PROGRAM Winder_data
VAR
	Power_lever_0: Power_lever;
	Clutch_0: Clutch;
	TP_0: TP;
	Brake_0: Brake;
	Standard_stuff_0:Standard_stuff;
	TP_1: TP;
	TP_2: TP;
END_VAR
VAR // added by the converter: edge detectors and wires of the graphical bodies
    _w1, _w2, _w3, _w4, _w5 : ANY;
END_VAR

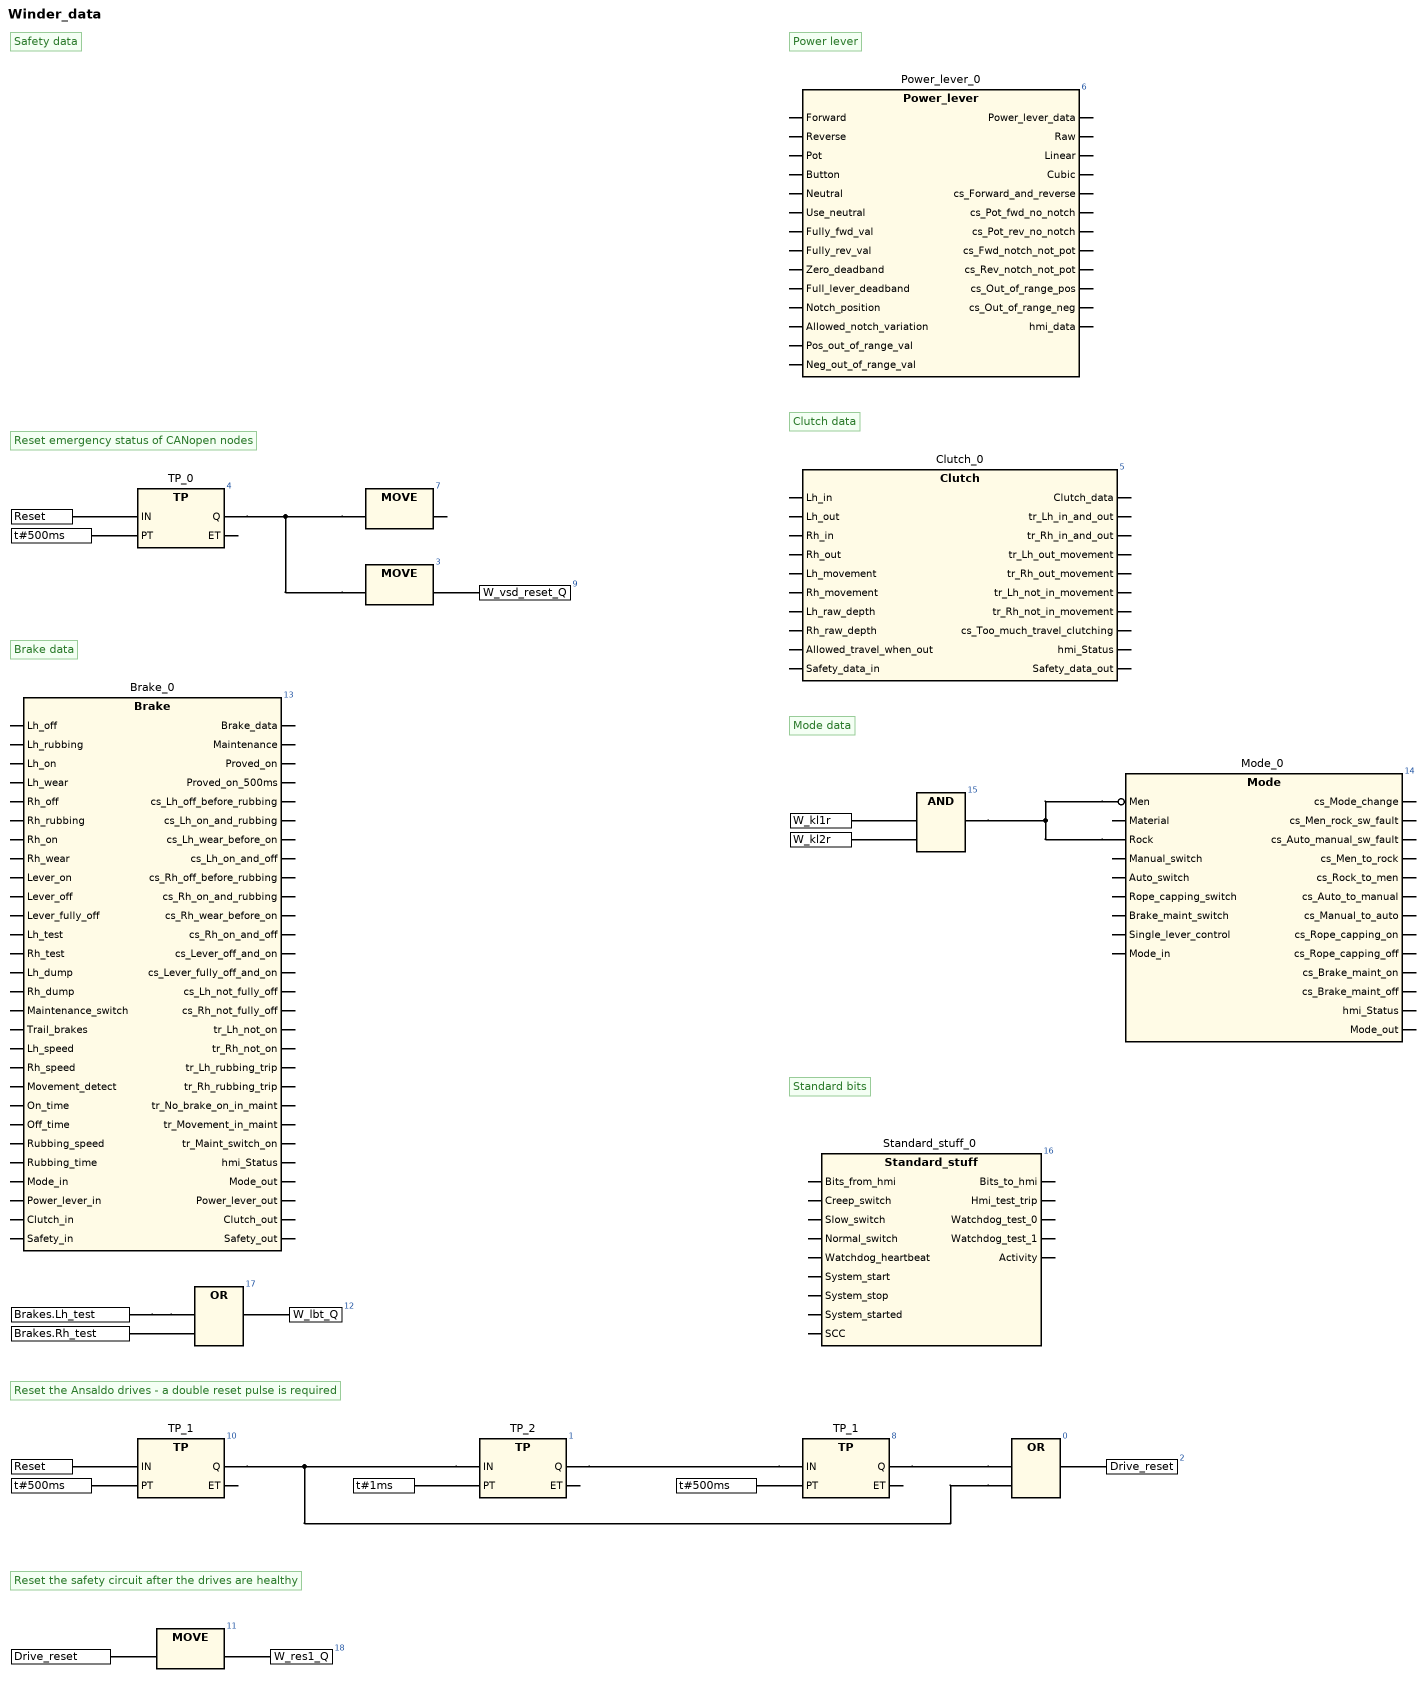
_w1 := TP_1.Q OR TP_1.Q;
TP_2(IN := TP_1.Q, PT := t#1ms); // TP
Drive_reset := _w1;
_w2 := TP_0.Q;
// Reset emergency status of CANopen nodes
TP_0(IN := Reset, PT := t#500ms); // TP
// Clutch data
Clutch_0(); // Clutch
// Safety data
// Power lever
Power_lever_0(); // Power_lever
(* TP_0.Q; result not used *)
TP_1(IN := TP_2.Q, PT := t#500ms); // TP
W_vsd_reset_Q := _w2;
// Reset the Ansaldo drives - a double reset pulse is required
TP_1(IN := Reset, PT := t#500ms); // TP
// Reset the safety circuit after the drives are healthy
_w3 := Drive_reset;
W_lbt_Q := _w4;
// Brake data
Brake_0(); // Brake
Mode_0(Men := NOT _w5, Rock := _w5); // Mode
// Mode data
_w5 := W_kl1r AND W_kl2r;
// Standard bits
Standard_stuff_0(); // Standard_stuff
_w4 := Brakes.Lh_test OR Brakes.Rh_test;
W_res1_Q := _w3;

METHOD Brake
VAR_INPUT
	Lh_off:BOOL;(*Left brake off signal - usually from left spring nest*)
	Lh_rubbing:BOOL; (*Left brake rubbing signal - usually from left spring nest*)
	Lh_on:BOOL; (*Left brake on signal - usually from left spring nest*)
	Lh_wear:BOOL; (*Left brake wear signal - usually from left spring nest*)
	Rh_off:BOOL; (*Right brake on signal - usually from right spring nest*)
	Rh_rubbing:BOOL; (*Right brake rubbing signal - usually from right spring nest*)
	Rh_on:BOOL; (*Right brake on signal - usually from right spring nest*)
	Rh_wear:BOOL; (*Right brake wear signal - usually from Right spring nest*)
	Lever_on:BOOL; (*Brake lever on limit switch*)
	Lever_off:BOOL; (*Brake lever off - normally from same limit switch as "Lever_on"*)
	Lever_fully_off:BOOL; (*Brake lever fully off limit switch. Necessary for automatic winders.*)
	Lh_test:BOOL; (*Left brake test switch - normally on driver's desk. Often the same switch as Lh_dump.*)
	Rh_test:BOOL; (*Right brake test switch - normally on driver's desk. Often the same switch as Rh_dump.*)
	Lh_dump:BOOL; (*Left brake dump switch - normally on driver's desk. Often the same switch as Lh_test.*)
	Rh_dump:BOOL; (*Right brake dump switch - normally on driver's desk. Often the same switch as Rh_test.*)
	Maintenance_switch:BOOL; (*Brake maintenance switch (can be on driver's desk or in control panels).*)
	Trail_brakes:BOOL; (*Trail brake control signal. Used to disable Lh_not_fully_off and Rh_not_fully_off trips.*)
	Lh_speed:INT; (*Left drum speed (normally in mm/s)*)
	Rh_speed:INT; (*Right drum speed (normally in mm/s)*)
	Movement_detect:BOOL; (*Drum movement detected (on either of the two drums in a double-drum winder)*)
	On_time:TIME; (*Maximum time allowed for brakes to apply.*)
	Off_time:TIME; (*Maximum time allowed for brakes to lift.*)
	Rubbing_speed:INT; (*Speed above which the brakes must be above the rubbing position*)
	Rubbing_time:TIME; (*Time before brake rubbing trips trigger *)
	Mode_in:dut_Mode;
	Power_lever_in:dut_Power_lever;
	Clutch_in:dut_Clutch;
	Safety_in:dut_Safety;
END_VAR
VAR_OUTPUT
	Brake_data:dut_Brake;
	Maintenance:BOOL; (*The winder is in brake maintenance mode*)
	Proved_on:BOOL; (*The brake lever (if in manual mode) and both brakes are on*)
	Proved_on_500ms:BOOL; (*The brakes have been proved on for 500ms*)
	cs_Lh_off_before_rubbing:BOOL; (*The Lh_off switch has closed but the Lh_rubbing switch has not yet closed*)
	cs_Lh_on_and_rubbing:BOOL; (*The Lh_on switch has closed but the Lh_rubbing switch is still closed*)
	cs_Lh_wear_before_on:BOOL; (*The Lh_on switch has closed but the Lh_rubbing switch is still closed*)
	cs_Lh_on_and_off:BOOL; (*The Lh_on and Lh_off switches are simultaneously closed*)
	cs_Rh_off_before_rubbing:BOOL; (*The Rh_off switch has closed but the Rh_rubbing switch has not yet closed*)
	cs_Rh_on_and_rubbing:BOOL; (*The Rh_on switch has closed but the Rh_rubbing switch is still closed*)
	cs_Rh_wear_before_on:BOOL; (*The Rh_on switch has closed but the Rh_rubbing switch is still closed*)
	cs_Rh_on_and_off:BOOL; (*The Rh_on and Rh_off switches are simultaneously closed*)
	cs_Lever_off_and_on:BOOL; (*The brake lever on and off switches are simultaneously closed*)
	cs_Lever_fully_off_and_on:BOOL; (*The brake lever on and fully off switches are simultaneously closed*)
	cs_Lh_not_fully_off:BOOL; (*The brake lever has been off for longer than the brake lift time but the Lh_off switch is not closed. Trail_brakes disables this fault.*)
	cs_Rh_not_fully_off:BOOL; (*The brake lever has been off for longer than the brake lift time but the Rh_off switch is not closed. Trail_brakes disables this fault.*)
	tr_Lh_not_on:BOOL; (*The brake lever has been on for longer than the brake application time but the Lh_on switch is not closed.*)
	tr_Rh_not_on:BOOL; (*The brake lever has been on for longer than the brake application time but the Rh_on switch is not closed.*)
	tr_Lh_rubbing_trip:BOOL; (*Lh_rubbing active above the rubbing trip speed*)
	tr_Rh_rubbing_trip:BOOL; (*Rh_rubbing active above the rubbing trip speed*)
	tr_No_brake_on_in_maint:BOOL; (*The power lever was moved from the neutral position in brake maintenance mode*)
	tr_Movement_in_maint:BOOL; (*Movement has been detected in brake maintenance mode*)
	tr_Maint_switch_on:BOOL; (*The brake maintenance switch is on but a brake is not dumped*)
	hmi_Status:ARRAY[1..2] OF WORD; (*Status bits for HMI*)
	Mode_out:dut_Mode;
	Power_lever_out:dut_Power_lever;
	Clutch_out:dut_Clutch;
	Safety_out:dut_Safety;
END_VAR
VAR
	TON_0: TON;
	Maintenance_req: BOOL;
	RS_0: RS;
	TON_1: TON;
	TON_2: TON;
	TON_3: TON;
	TON_4: TON;
	TON_5: TON;
	TON_6: TON;
	TON_7: TON;
	TON_8: TON;
	TON_9: TON;
	TON_10: TON;
	TON_11: TON;
	TON_12: TON;
	TON_13: TON;
	TON_14: TON;
	TON_15: TON;
	TON_16: TON;
	TON_17: TON;
END_VAR
VAR_INST // added by the converter: edge detectors and wires of the graphical bodies
    _w1, _w3, _w5, _w8, _w9, _w10, _w11, _w12, _w13, _w14, _w15, _w16, _w17, _w18, _w19, _w20, _w21, _w22, _w23, _w24, _w26, _w27, _w28 : BOOL;
    _w2, _w4, _w6, _w7, _w25 : ANY;
END_VAR
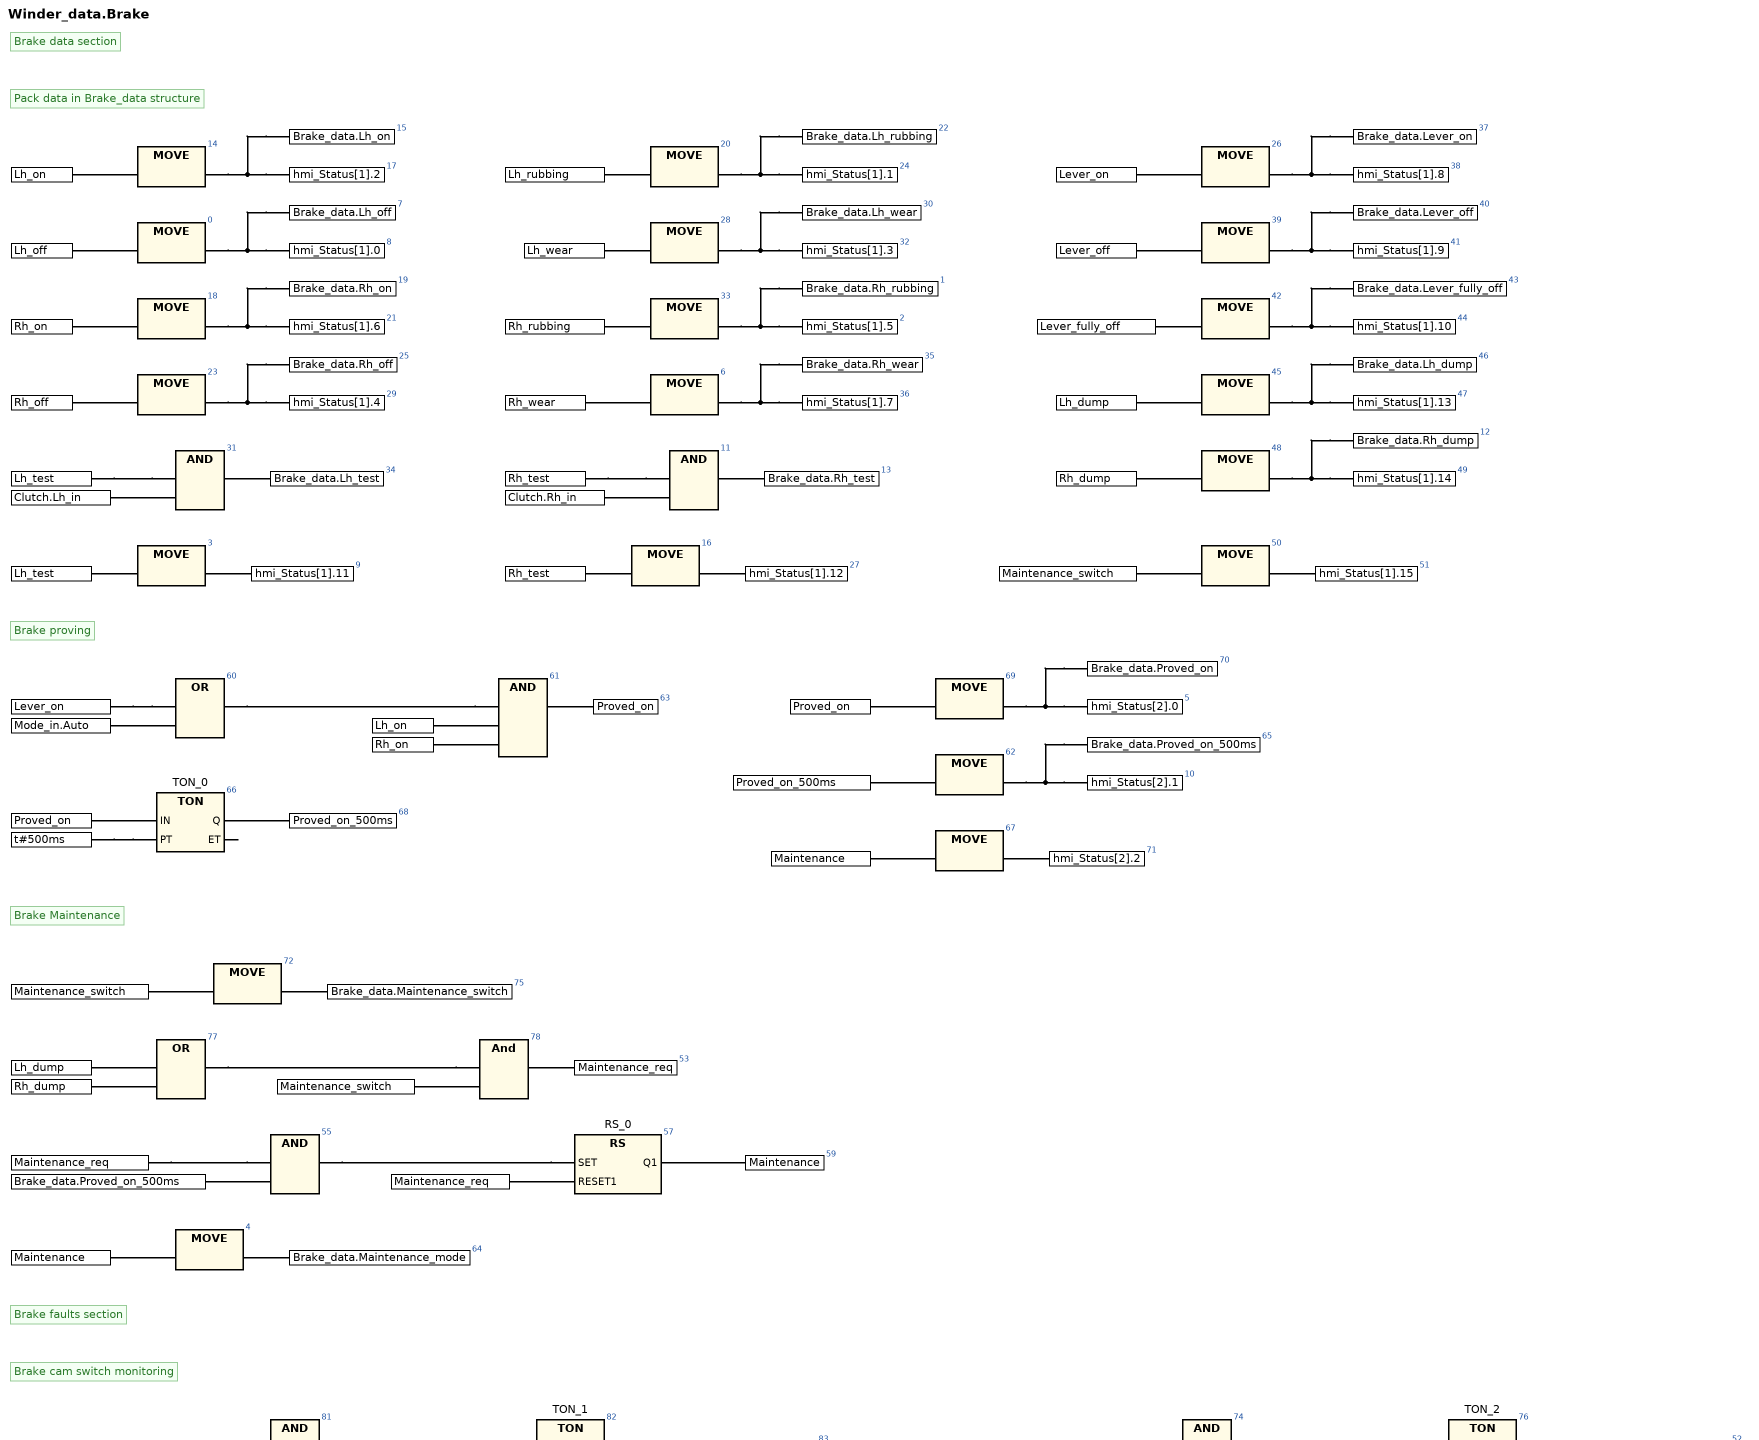
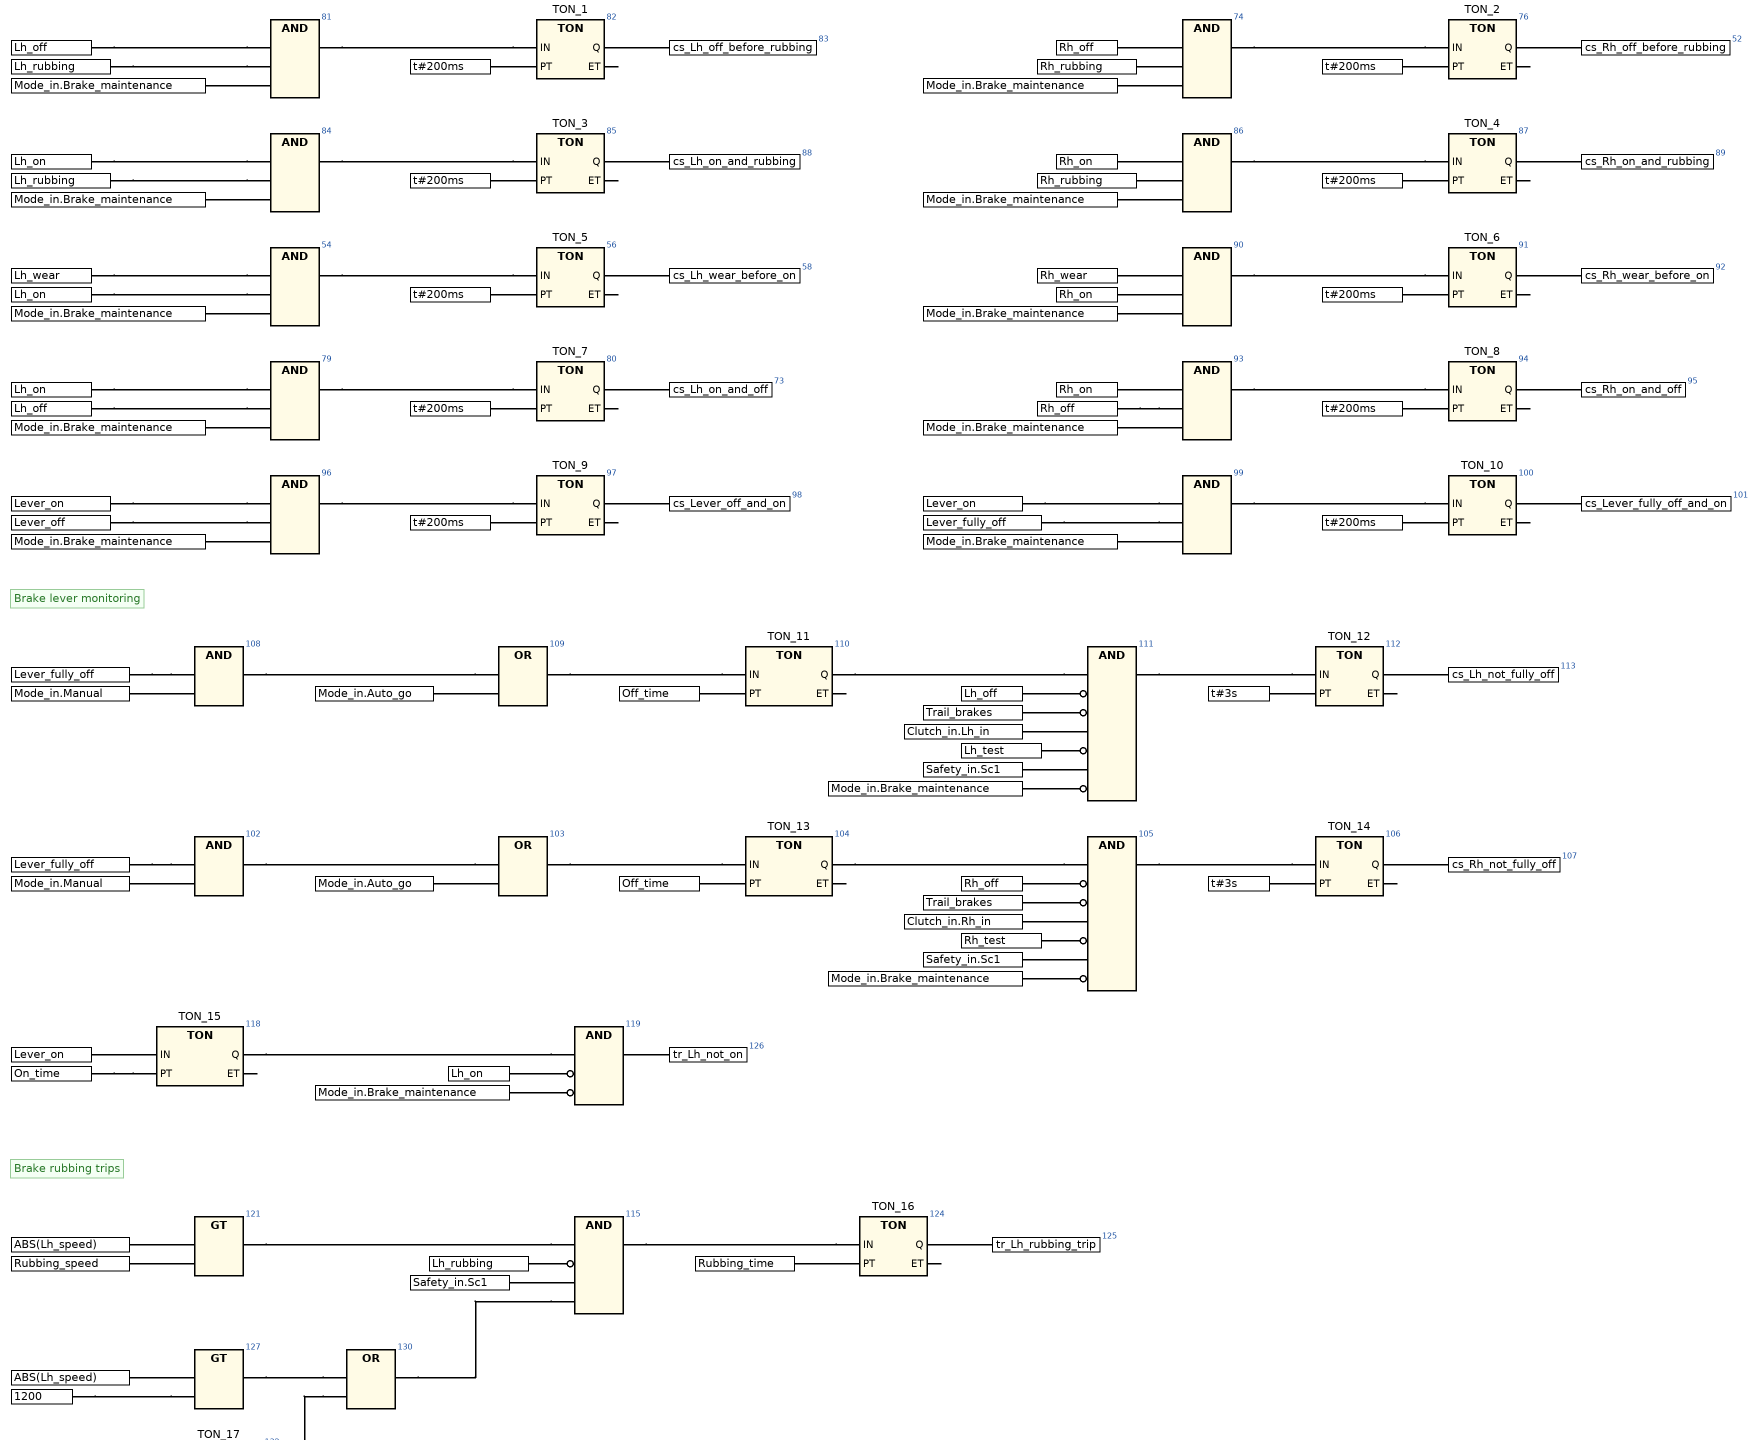
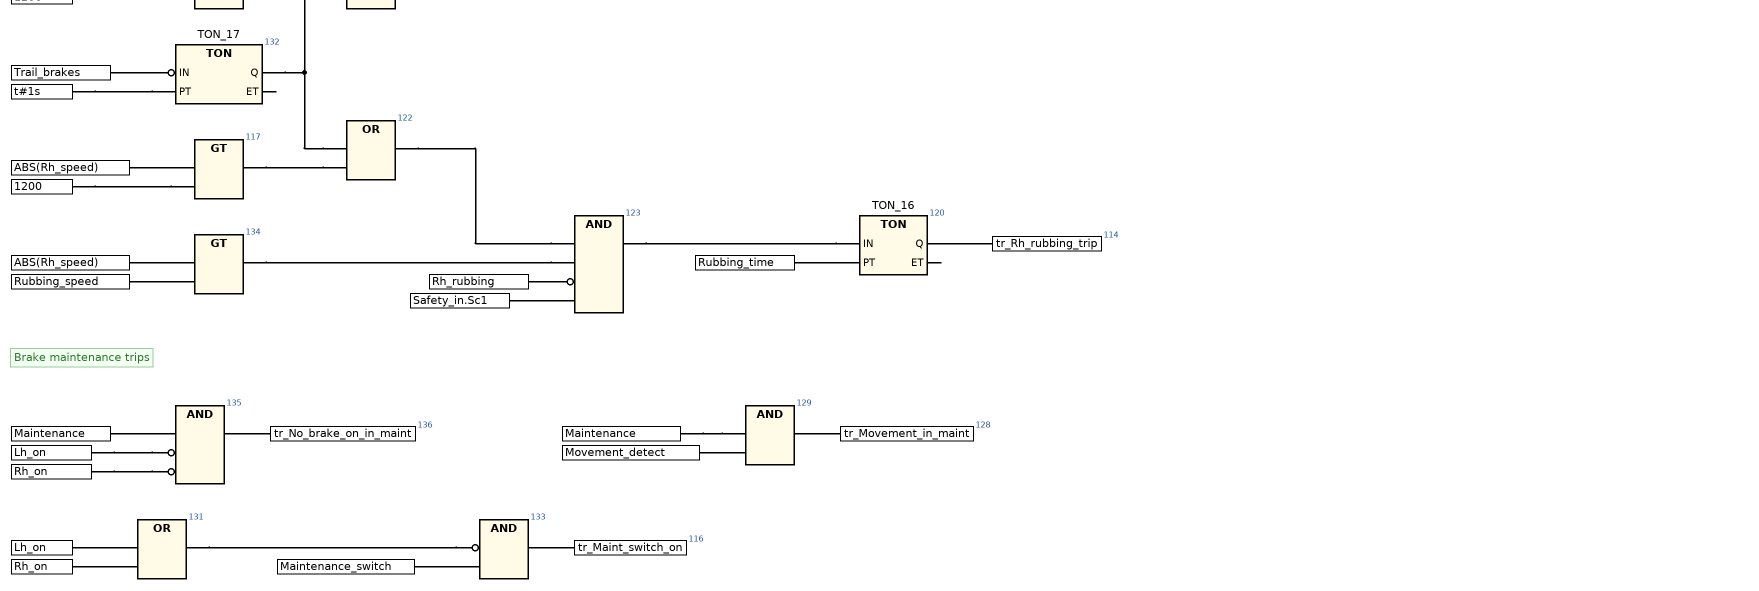
_w1 := Lh_off;
Brake_data.Rh_rubbing := _w2;
hmi_Status[1].5 := _w2;
_w3 := Maintenance;
hmi_Status[2].0 := _w4;
_w5 := Rh_wear;
Brake_data.Lh_off := _w1;
hmi_Status[1].0 := _w1;
hmi_Status[1].11 := Lh_test;
hmi_Status[2].1 := _w6;
Brake_data.Rh_dump := _w7;
Brake_data.Rh_test := Rh_test AND Clutch.Rh_in;
// Brake data section
// Pack data in Brake_data structure
_w8 := Lh_on;
Brake_data.Lh_on := _w8;
hmi_Status[1].2 := _w8;
_w9 := Rh_on;
Brake_data.Rh_on := _w9;
_w10 := Lh_rubbing;
hmi_Status[1].6 := _w9;
Brake_data.Lh_rubbing := _w10;
_w11 := Rh_off;
hmi_Status[1].1 := _w10;
Brake_data.Rh_off := _w11;
_w12 := Lever_on;
hmi_Status[1].12 := Rh_test;
_w13 := Lh_wear;
hmi_Status[1].4 := _w11;
Brake_data.Lh_wear := _w13;
hmi_Status[1].3 := _w13;
_w2 := Rh_rubbing;
Brake_data.Lh_test := Lh_test AND Clutch.Lh_in;
Brake_data.Rh_wear := _w5;
hmi_Status[1].7 := _w5;
Brake_data.Lever_on := _w12;
hmi_Status[1].8 := _w12;
_w14 := Lever_off;
Brake_data.Lever_off := _w14;
hmi_Status[1].9 := _w14;
_w15 := Lever_fully_off;
Brake_data.Lever_fully_off := _w15;
hmi_Status[1].10 := _w15;
_w16 := Lh_dump;
Brake_data.Lh_dump := _w16;
hmi_Status[1].13 := _w16;
_w7 := Rh_dump;
hmi_Status[1].14 := _w7;
hmi_Status[1].15 := Maintenance_switch;
cs_Rh_off_before_rubbing := TON_2.Q;
Maintenance_req := _w17;
_w18 := Maintenance_req AND Brake_data.Proved_on_500ms;
TON_5(IN := Lh_wear AND Lh_on AND Mode_in.Brake_maintenance, PT := t#200ms); // TON
RS_0(SET := _w18, RESET1 := Maintenance_req); // RS
cs_Lh_wear_before_on := TON_5.Q;
Maintenance := RS_0.Q1;
// Brake proving
_w6 := Proved_on_500ms;
Proved_on := (Lever_on OR Mode_in.Auto) AND Lh_on AND Rh_on;
Brake_data.Maintenance_mode := _w3;
Brake_data.Proved_on_500ms := _w6;
TON_0(IN := Proved_on, PT := t#500ms); // TON
Proved_on_500ms := TON_0.Q;
_w4 := Proved_on;
Brake_data.Proved_on := _w4;
hmi_Status[2].2 := Maintenance;
// Brake Maintenance
cs_Lh_on_and_off := TON_7.Q;
Brake_data.Maintenance_switch := Maintenance_switch;
TON_2(IN := Rh_off AND Rh_rubbing AND Mode_in.Brake_maintenance, PT := t#200ms); // TON
_w17 := (Lh_dump OR Rh_dump) AND Maintenance_switch;
TON_7(IN := Lh_on AND Lh_off AND Mode_in.Brake_maintenance, PT := t#200ms); // TON
// Brake faults section
// Brake cam switch monitoring
TON_1(IN := Lh_off AND Lh_rubbing AND Mode_in.Brake_maintenance, PT := t#200ms); // TON
cs_Lh_off_before_rubbing := TON_1.Q;
TON_3(IN := Lh_on AND Lh_rubbing AND Mode_in.Brake_maintenance, PT := t#200ms); // TON
TON_4(IN := Rh_on AND Rh_rubbing AND Mode_in.Brake_maintenance, PT := t#200ms); // TON
cs_Lh_on_and_rubbing := TON_3.Q;
cs_Rh_on_and_rubbing := TON_4.Q;
TON_6(IN := Rh_wear AND Rh_on AND Mode_in.Brake_maintenance, PT := t#200ms); // TON
cs_Rh_wear_before_on := TON_6.Q;
TON_8(IN := Rh_on AND Rh_off AND Mode_in.Brake_maintenance, PT := t#200ms); // TON
cs_Rh_on_and_off := TON_8.Q;
TON_9(IN := Lever_on AND Lever_off AND Mode_in.Brake_maintenance, PT := t#200ms); // TON
cs_Lever_off_and_on := TON_9.Q;
TON_10(IN := Lever_on AND Lever_fully_off AND Mode_in.Brake_maintenance, PT := t#200ms); // TON
cs_Lever_fully_off_and_on := TON_10.Q;
TON_13(IN := Lever_fully_off AND Mode_in.Manual OR Mode_in.Auto_go, PT := Off_time); // TON
TON_14(IN := TON_13.Q AND NOT Rh_off AND NOT Trail_brakes AND Clutch_in.Rh_in AND NOT Rh_test AND Safety_in.Sc1 AND NOT Mode_in.Brake_maintenance, PT := t#3s); // TON
cs_Rh_not_fully_off := TON_14.Q;
// Brake lever monitoring
TON_11(IN := Lever_fully_off AND Mode_in.Manual OR Mode_in.Auto_go, PT := Off_time); // TON
TON_12(IN := TON_11.Q AND NOT Lh_off AND NOT Trail_brakes AND Clutch_in.Lh_in AND NOT Lh_test AND Safety_in.Sc1 AND NOT Mode_in.Brake_maintenance, PT := t#3s); // TON
cs_Lh_not_fully_off := TON_12.Q;
tr_Rh_rubbing_trip := TON_16.Q;
_w21 := _w19 AND NOT Lh_rubbing AND Safety_in.Sc1 AND _w20;
tr_Maint_switch_on := _w22;
_w23 := (ABS(Rh_speed)) > 1200;
TON_15(IN := Lever_on, PT := On_time); // TON
_w24 := TON_15.Q AND NOT Lh_on AND NOT Mode_in.Brake_maintenance;
TON_16(IN := _w25, PT := Rubbing_time); // TON
// Brake rubbing trips
_w19 := (ABS(Lh_speed)) > Rubbing_speed;
_w25 := (TON_17.Q OR _w23) AND _w26 AND NOT Rh_rubbing AND Safety_in.Sc1;
TON_16(IN := _w21, PT := Rubbing_time); // TON
tr_Lh_rubbing_trip := TON_16.Q;
tr_Lh_not_on := _w24;
tr_Movement_in_maint := _w27;
_w27 := Maintenance AND Movement_detect;
_w20 := (ABS(Lh_speed)) > 1200 OR TON_17.Q;
_w28 := Lh_on OR Rh_on;
TON_17(IN := NOT Trail_brakes, PT := t#1s); // TON
_w22 := NOT _w28 AND Maintenance_switch;
_w26 := (ABS(Rh_speed)) > Rubbing_speed;
// Brake maintenance trips
tr_No_brake_on_in_maint := Maintenance AND NOT Lh_on AND NOT Rh_on;
END_METHOD

METHOD Clutch
VAR_INPUT
	Lh_in:BOOL; (*Left hand clutch in switch*)
	Lh_out:BOOL; (*Left hand clutch out switch*)
	Rh_in:BOOL; (*Right hand clutch in switch*)
	Rh_out:BOOL; (*Right hand clutch out switch*)
	Lh_movement:BOOL; (*Movement on left hand drum*)
	Rh_movement:BOOL; (*Movement on right hand drum*)
	Lh_raw_depth:DINT; (*Left conveyance raw depth*)
	Rh_raw_depth:DINT; (*Right conveyance raw depth*)
	Allowed_travel_when_out:DINT; (*Amount of travel allowed while engaging/disengaging a clutch*)
	Safety_data_in:dut_Safety; (*Data structure with safety and reset data*)
END_VAR
VAR_OUTPUT
	Clutch_data:dut_Clutch; (*Clutch data structure*)
	tr_Lh_in_and_out:BOOL; (*Left hand clutch in and out switches both energised*)
	tr_Rh_in_and_out:BOOL; (*Right hand clutch in and out switches both energised*)
	tr_Lh_out_movement:BOOL; (*Movement was detected on the left hand drum when the left clutch was out*)
	tr_Rh_out_movement:BOOL; (*Movement was detected on the right hand drum when the right clutch was out*)
	tr_Lh_not_in_movement:BOOL; (*Movement was detected on the left hand drum when the left clutch was not in*)
	tr_Rh_not_in_movement:BOOL; (*Movement was detected on the right hand drum when the right clutch was not in*)
	cs_Too_much_travel_clutching:BOOL; (*There was too much drum travel while engaging/disengaging a clutch*)
	hmi_Status:WORD; (*Status bits for HMI*)
	Safety_data_out:dut_Safety; (*Data structure with safety and reset data*)
END_VAR
VAR
	TON_0: TON;
	TON_1: TON;
	TON_2: TON;
	TON_3: TON;
	Lh_start_depth: DINT;
	RS_0: RS;
	Rh_start_depth: DINT;
	RS_1: RS;
END_VAR
VAR_INST // added by the converter: edge detectors and wires of the graphical bodies
    _w1, _w2, _w3, _w4, _w5, _w8, _w12 : ANY;
    _w6, _w7, _w9, _w10 : BOOL;
    _w11, _w13 : DINT;
END_VAR
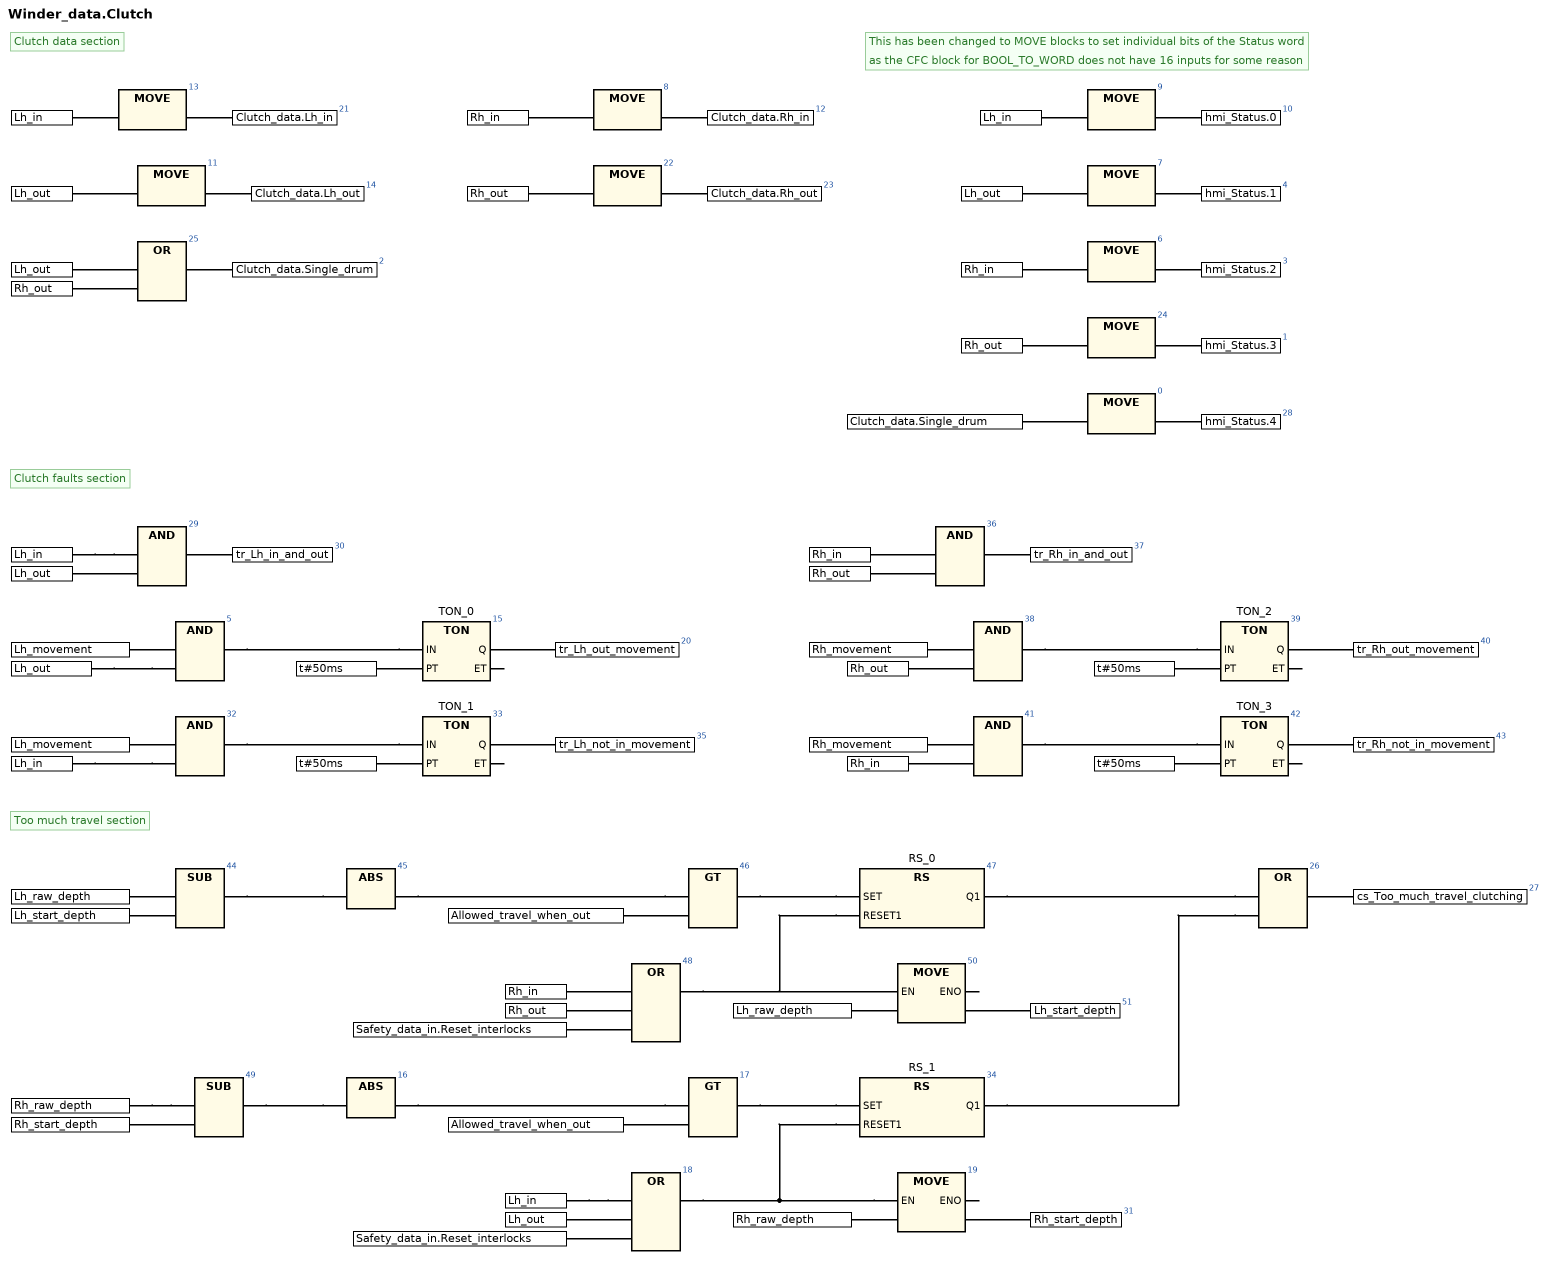
_w1 := Clutch_data.Single_drum;
hmi_Status.3 := _w2;
Clutch_data.Single_drum := _w3;
hmi_Status.2 := _w4;
hmi_Status.1 := _w5;
_w6 := Lh_movement AND Lh_out;
_w4 := Rh_in;
_w5 := Lh_out;
// This has been changed to MOVE blocks to set individual bits of the Status word
// as the CFC block for BOOL_TO_WORD does not have 16 inputs for some reason
hmi_Status.0 := Lh_in;
Clutch_data.Rh_in := Rh_in;
// Clutch data section
_w7 := Lh_in;
Clutch_data.Lh_out := Lh_out;
TON_0(IN := _w6, PT := t#50ms); // TON
_w9 := ABS(_w8) > Allowed_travel_when_out;
_w10 := Lh_in OR Lh_out OR Safety_data_in.Reset_interlocks;
IF _w10 THEN _w11 := Rh_raw_depth; END_IF
tr_Lh_out_movement := TON_0.Q;
Clutch_data.Lh_in := _w7;
Clutch_data.Rh_out := Rh_out;
_w2 := Rh_out;
_w3 := Lh_out OR Rh_out;
cs_Too_much_travel_clutching := RS_0.Q1 OR RS_1.Q1;
hmi_Status.4 := _w1;
// Clutch faults section
tr_Lh_in_and_out := Lh_in AND Lh_out;
Rh_start_depth := _w11;
TON_1(IN := Lh_movement AND Lh_in, PT := t#50ms); // TON
RS_1(SET := _w9, RESET1 := _w10); // RS
tr_Lh_not_in_movement := TON_1.Q;
tr_Rh_in_and_out := Rh_in AND Rh_out;
TON_2(IN := Rh_movement AND Rh_out, PT := t#50ms); // TON
tr_Rh_out_movement := TON_2.Q;
TON_3(IN := Rh_movement AND Rh_in, PT := t#50ms); // TON
tr_Rh_not_in_movement := TON_3.Q;
// Too much travel section
RS_0(SET := ABS(Lh_raw_depth - Lh_start_depth) > Allowed_travel_when_out, RESET1 := _w12); // RS
_w12 := Rh_in OR Rh_out OR Safety_data_in.Reset_interlocks;
_w8 := Rh_raw_depth - Rh_start_depth;
IF _w12 THEN _w13 := Lh_raw_depth; END_IF
Lh_start_depth := _w13;
END_METHOD

METHOD Mode
VAR_INPUT
	Men:BOOL;
	Material:BOOL;
	Rock:BOOL;
	Manual_switch:BOOL;
	Auto_switch:BOOL;
	Rope_capping_switch:BOOL;
	Brake_maint_switch:BOOL;
	Single_lever_control:BOOL;
	Mode_in:dut_Mode;
END_VAR
VAR_OUTPUT
	cs_Mode_change:BOOL;
	cs_Men_rock_sw_fault:BOOL;
	cs_Auto_manual_sw_fault:BOOL;
	cs_Men_to_rock:BOOL;
	cs_Rock_to_men:BOOL;
	cs_Auto_to_manual:BOOL;
	cs_Manual_to_auto:BOOL;
	cs_Rope_capping_on:BOOL;
	cs_Rope_capping_off:BOOL;
	cs_Brake_maint_on:BOOL;
	cs_Brake_maint_off:BOOL;
	hmi_Status:WORD;
	Mode_out:dut_Mode;
END_VAR

VAR
	F_TRIG_0: F_TRIG;
	R_TRIG_0: R_TRIG;
	R_TRIG_1: R_TRIG;
	F_TRIG_1: F_TRIG;
	R_TRIG_2: R_TRIG;
	F_TRIG_2: F_TRIG;
	R_TRIG_3: R_TRIG;
	F_TRIG_3: F_TRIG;
	R_TRIG_4: R_TRIG;
	F_TRIG_4: F_TRIG;
	R_TRIG_5: R_TRIG;
	F_TRIG_5: F_TRIG;
	TON_0: TON;
END_VAR
VAR_INST // added by the converter: edge detectors and wires of the graphical bodies
    _w1, _w2, _w5, _w6, _w9, _w10, _w12, _w13, _w15, _w16, _w17 : BOOL;
    _w3, _w4, _w7, _w8, _w11, _w14 : ANY;
END_VAR
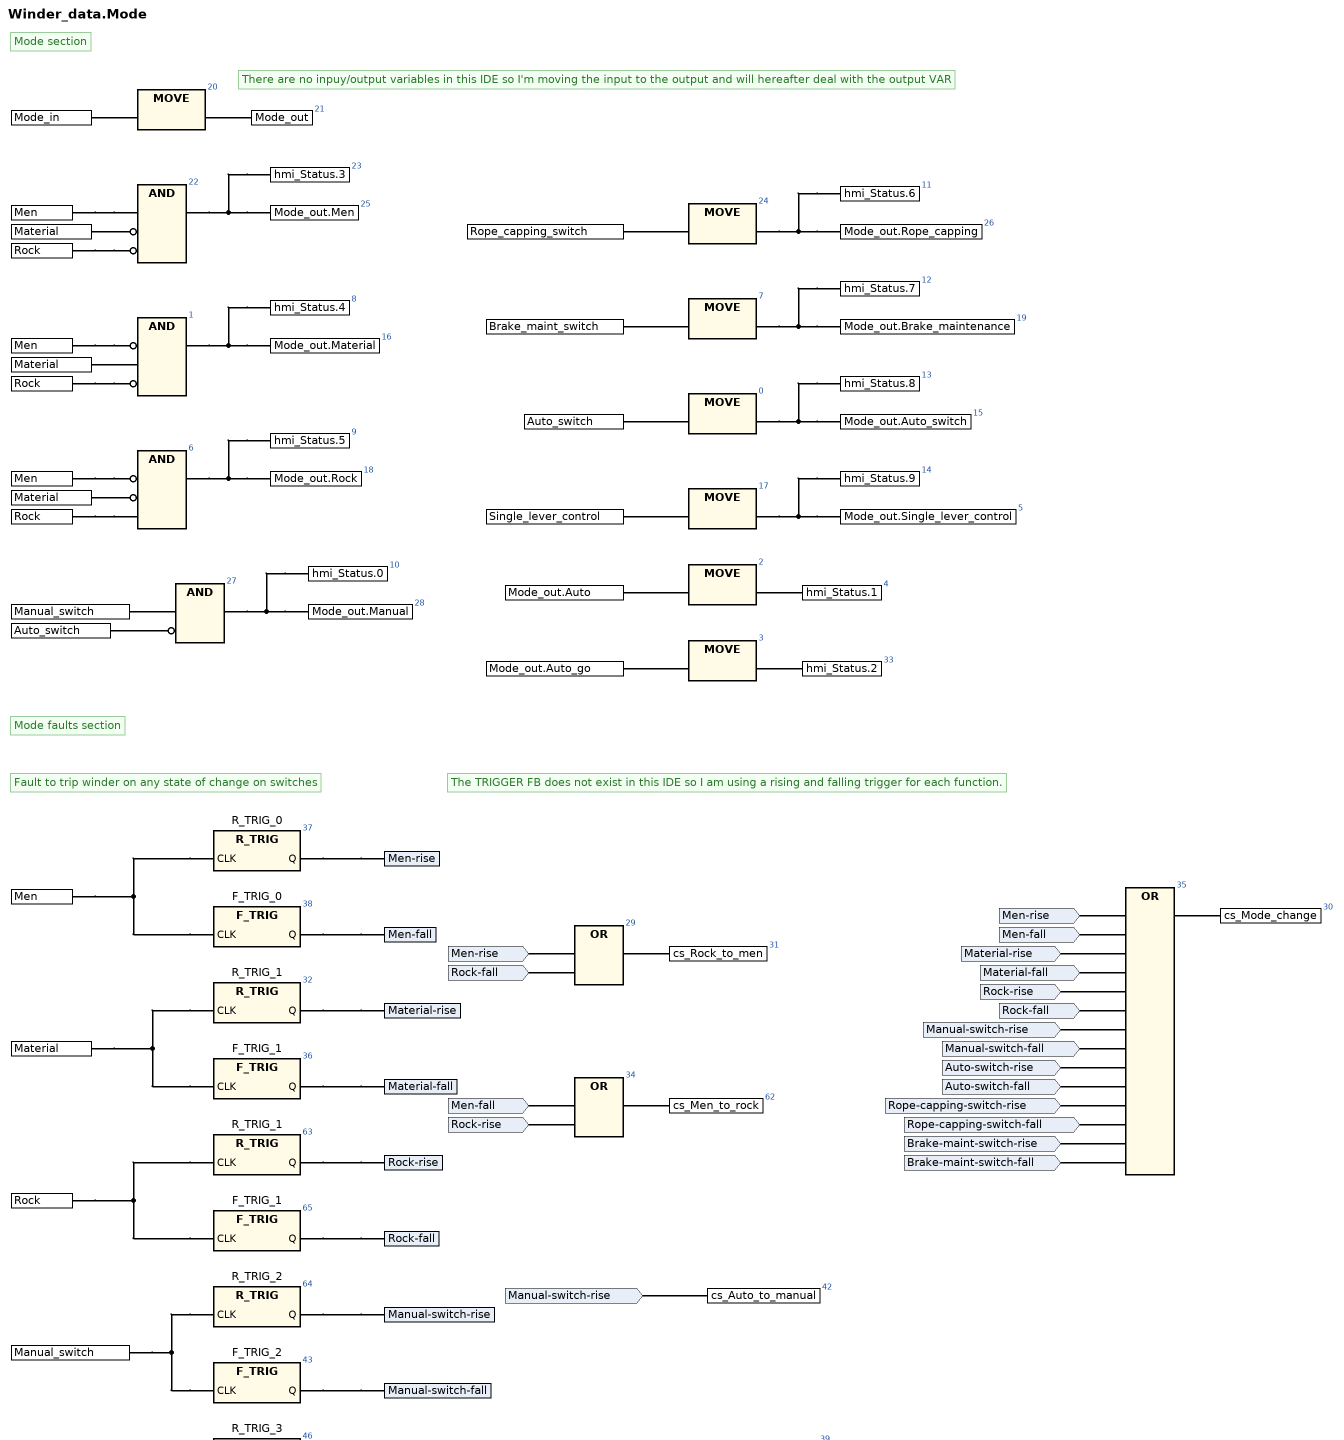
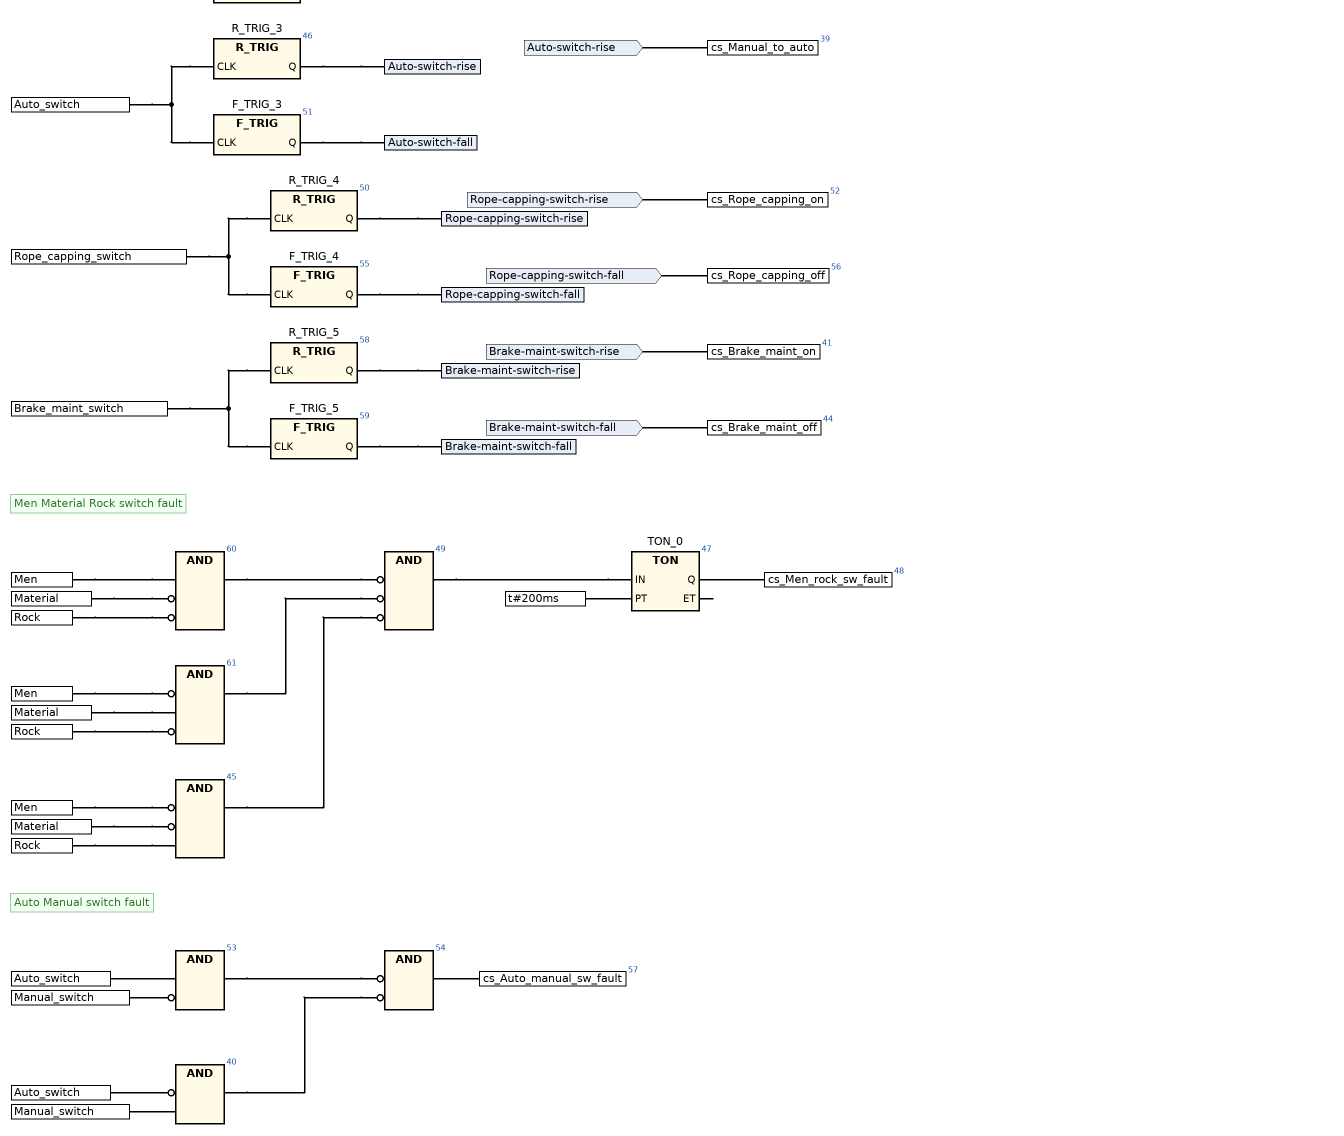
_w1 := Auto_switch;
_w2 := NOT Men AND Material AND NOT Rock;
_w3 := Mode_out.Auto_go;
hmi_Status.1 := Mode_out.Auto;
Mode_out.Single_lever_control := _w4;
_w5 := NOT Men AND NOT Material AND Rock;
_w6 := Brake_maint_switch;
hmi_Status.4 := _w2;
hmi_Status.5 := _w5;
hmi_Status.0 := _w7;
hmi_Status.6 := _w8;
hmi_Status.7 := _w6;
hmi_Status.8 := _w1;
hmi_Status.9 := _w4;
Mode_out.Auto_switch := _w1;
Mode_out.Material := _w2;
_w4 := Single_lever_control;
Mode_out.Rock := _w5;
Mode_out.Brake_maintenance := _w6;
// Mode section
// There are no inpuy/output variables in this IDE so I'm moving the input to the output and will hereafter deal with the output VAR
Mode_out := Mode_in;
_w9 := Men AND NOT Material AND NOT Rock;
hmi_Status.3 := _w9;
_w8 := Rope_capping_switch;
Mode_out.Men := _w9;
Mode_out.Rope_capping := _w8;
_w7 := Manual_switch AND NOT Auto_switch;
Mode_out.Manual := _w7;
cs_Mode_change := _w10;
cs_Rock_to_men := R_TRIG_0.Q OR F_TRIG_1.Q;
R_TRIG_1(CLK := Material); // R_TRIG
hmi_Status.2 := _w3;
_w11 := F_TRIG_0.Q OR R_TRIG_1.Q;
_w10 := R_TRIG_0.Q OR F_TRIG_0.Q OR R_TRIG_1.Q OR F_TRIG_1.Q OR R_TRIG_1.Q OR F_TRIG_1.Q OR R_TRIG_2.Q OR F_TRIG_2.Q OR R_TRIG_3.Q OR F_TRIG_3.Q OR R_TRIG_4.Q OR F_TRIG_4.Q OR R_TRIG_5.Q OR F_TRIG_5.Q;
F_TRIG_1(CLK := Material); // F_TRIG
// Mode faults section
// Fault to trip winder on any state of change on switches
// The TRIGGER FB does not exist in this IDE so I am using a rising and falling trigger for each function.
R_TRIG_0(CLK := Men); // R_TRIG
F_TRIG_0(CLK := Men); // F_TRIG
cs_Manual_to_auto := R_TRIG_3.Q;
_w12 := NOT Auto_switch AND Manual_switch;
cs_Brake_maint_on := R_TRIG_5.Q;
cs_Auto_to_manual := R_TRIG_2.Q;
F_TRIG_2(CLK := Manual_switch); // F_TRIG
cs_Brake_maint_off := F_TRIG_5.Q;
_w13 := NOT Men AND NOT Material AND Rock;
R_TRIG_3(CLK := Auto_switch); // R_TRIG
TON_0(IN := _w14, PT := t#200ms); // TON
cs_Men_rock_sw_fault := TON_0.Q;
_w14 := NOT _w15 AND NOT _w16 AND NOT _w13;
R_TRIG_4(CLK := Rope_capping_switch); // R_TRIG
F_TRIG_3(CLK := Auto_switch); // F_TRIG
cs_Rope_capping_on := R_TRIG_4.Q;
// Auto Manual switch fault
_w17 := NOT (Auto_switch AND NOT Manual_switch) AND NOT _w12;
F_TRIG_4(CLK := Rope_capping_switch); // F_TRIG
cs_Rope_capping_off := F_TRIG_4.Q;
cs_Auto_manual_sw_fault := _w17;
R_TRIG_5(CLK := Brake_maint_switch); // R_TRIG
F_TRIG_5(CLK := Brake_maint_switch); // F_TRIG
// Men Material Rock switch fault
_w15 := Men AND NOT Material AND NOT Rock;
_w16 := NOT Men AND Material AND NOT Rock;
cs_Men_to_rock := _w11;
R_TRIG_1(CLK := Rock); // R_TRIG
R_TRIG_2(CLK := Manual_switch); // R_TRIG
F_TRIG_1(CLK := Rock); // F_TRIG
END_METHOD

METHOD Power_lever
VAR_INPUT
	Forward:BOOL; (*Lever notch 1 forward*)
	Reverse:BOOL; (*Lever notch 1 reverse*)
	Pot:INT; (*Analogue value from lever potentiometer*)
	Button:BOOL;
	Neutral:BOOL; 
	Use_neutral:BOOL;
	Fully_fwd_val:INT; (*Value of analogue input when lever is fully forward*)
	Fully_rev_val:INT; (*Value of analogue input when lever is fully reverse*)
	Zero_deadband:INT; (*Lever zero position deadband on a scale of 0 to 10 000 i.e. a value of 100 gives a 1% deadband in each direction*)
	Full_lever_deadband:INT; (*Lever fully forward or reverse deadband on a scale of 0 to 10 000 i.e. a value of 100 gives a 1% deadband*)
	Notch_position:INT; (*Lever value (-10 000 to 10 000, no deadbands) at which forward and reverse notches change state*)
	Allowed_notch_variation:INT; (*Allowed variation in notch position*)
	Pos_out_of_range_val:INT; (*If the analogue Pot value exceeds this threshold, a fault will be generated.*)
	Neg_out_of_range_val:INT; (*If the analogue Pot value is less than this threshold, a fault will be generated.*)
END_VAR
VAR_OUTPUT
	Power_lever_data:dut_Power_lever; (*Power lever data packed into a single structure.*)
	Raw:INT; (*Linear scaled lever value with no deadbands applied. -10 000 = fully reverse. +10 000 = fully forward.*)
	Linear:INT; (*Linear scaled lever value with deadbands applied. -10 000 = fully reverse. +10 000 = fully forward.*)
	Cubic:INT; (*Cubic scaling applied to lever value with deadbands applied. -10 000 = fully reverse. +10 000 = fully forward.*)
	cs_Forward_and_reverse:BOOL; (*Forward and reverse inputs both energised.*)
	cs_Pot_fwd_no_notch:BOOL; (*Pot shows that lever is forward but the forward notch is not activated*)
	cs_Pot_rev_no_notch:BOOL; (*Pot shows that lever is reverse but the reverse notch is not activated*)
	cs_Fwd_notch_not_pot:BOOL; (*Reverse notch is activated but the pot does not show that the lever is past the reverse notch*)
	cs_Rev_notch_not_pot:BOOL; (*Forward notch is activated but the pot does not show that the lever is past the forward notch*)
	cs_Out_of_range_pos:BOOL; (*The Pot value is out of range in the positive direction*)
	cs_Out_of_range_neg:BOOL; (*The Pot value is out of range in the negative direction*)
	hmi_data:dut_hmi_Power_lever; (*HMI status bits as well as Raw, Linear and Cubic values*)
END_VAR
VAR_IN_OUT
	Test: INT;
END_VAR
VAR
	Linear_abs: INT;
	hmi_Word:WORD;
	TON_0: TON;
	TON_2: TON;
	TON_1: TON;
	TON_3: TON;
END_VAR
VAR_INST // added by the converter: edge detectors and wires of the graphical bodies
    _w1, _w2, _w10 : REAL;
    _w3, _w4, _w5, _w11, _w13, _w14, _w15, _w16, _w22, _w24, _w25 : ANY;
    _w6, _w7, _w8, _w9, _w21 : INT;
    _w12, _w17, _w18, _w19, _w20, _w23 : BOOL;
END_VAR
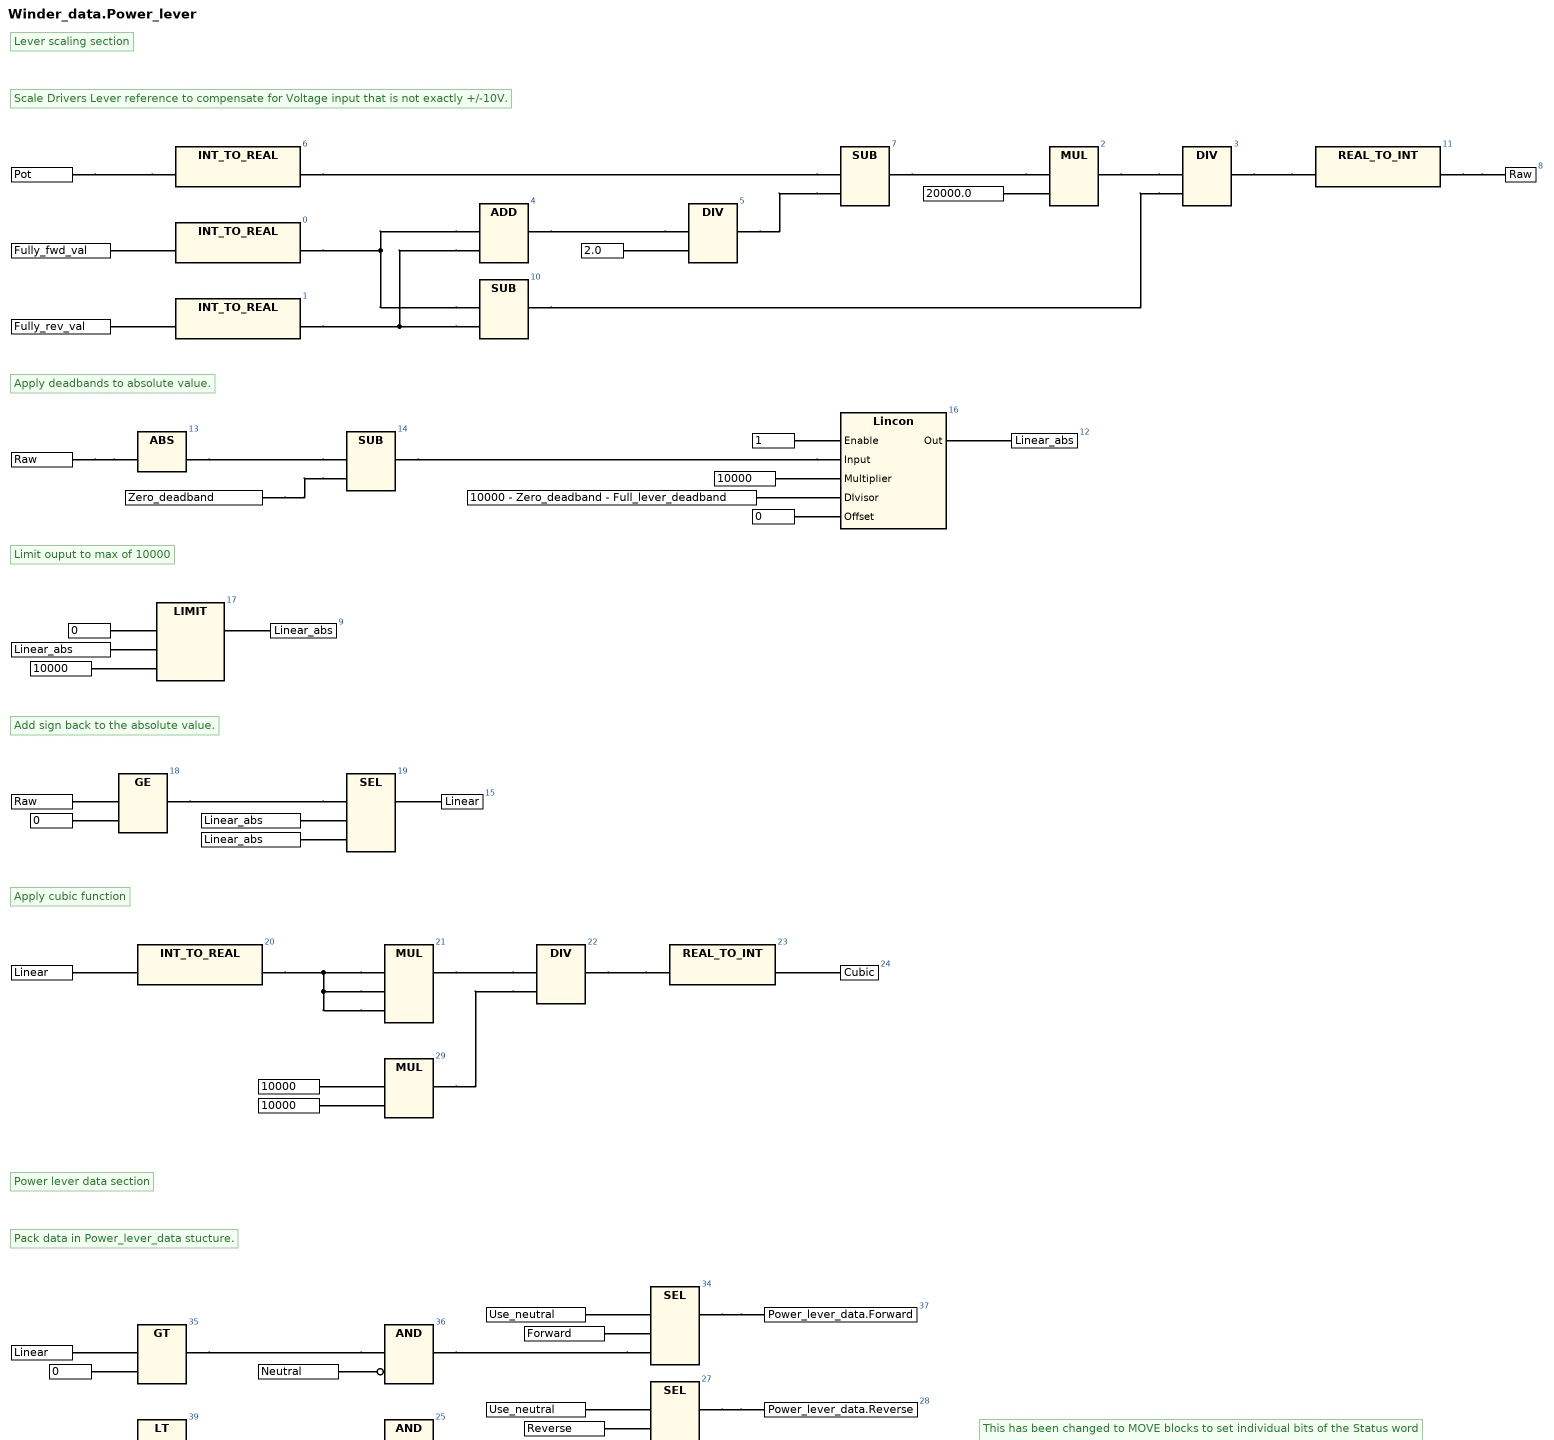
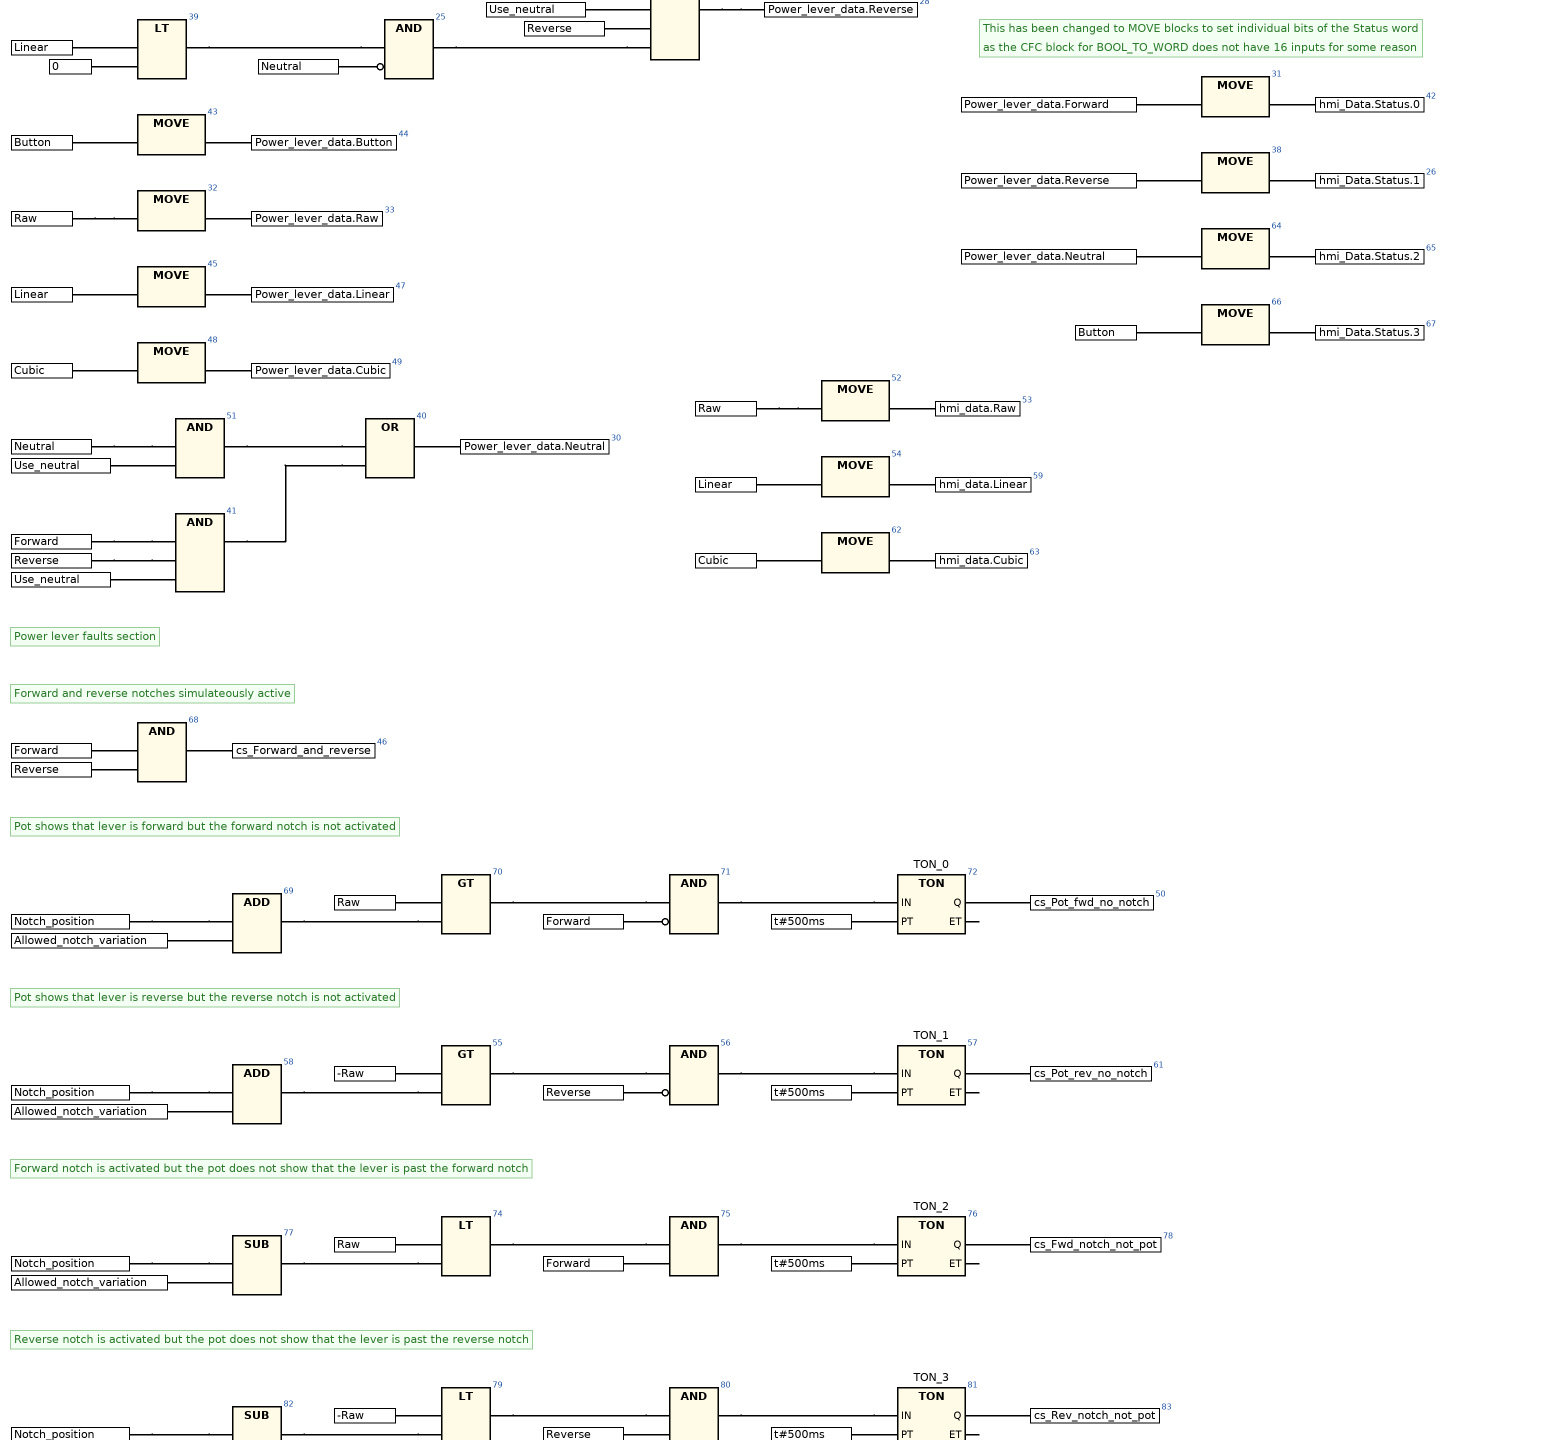
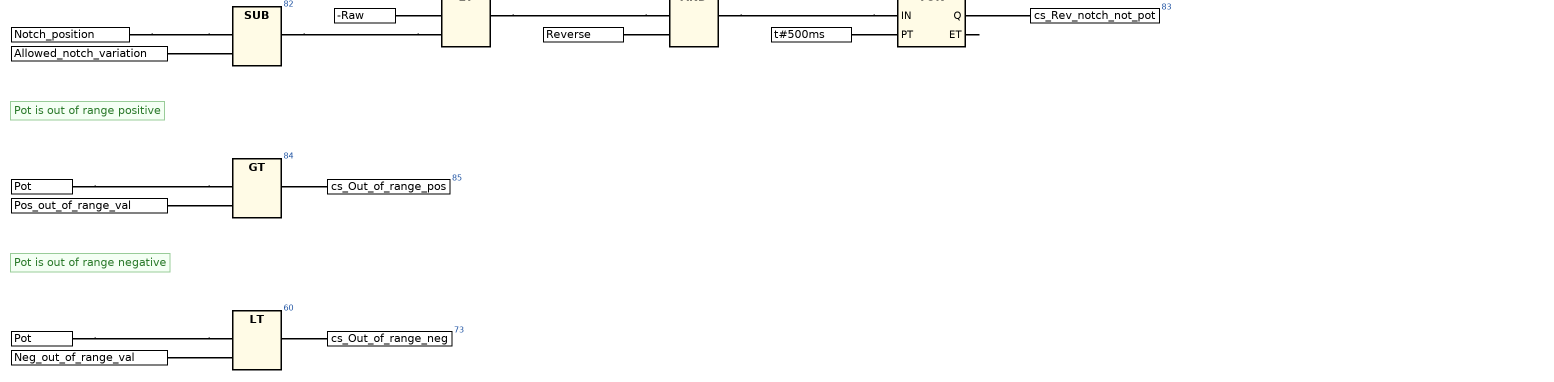
_w1 := INT_TO_REAL(Fully_fwd_val);
_w2 := INT_TO_REAL(Fully_rev_val);
_w5 := (_w3 * 20000.0) / _w4;
// Lever scaling section
// Scale Drivers Lever reference to compensate for Voltage input that is not exactly +/-10V.
_w3 := INT_TO_REAL(Pot) - (_w1 + _w2) / 2.0;
Raw := _w6;
Linear_abs := _w7;
_w4 := _w1 - _w2;
_w6 := REAL_TO_INT(_w5);
Linear_abs := _w8;
// Apply deadbands to absolute value.
Linear := _w9;
_w8 := Lincon(Enable := 1, Input := ABS(Raw) - Zero_deadband, Multiplier := 10000, DIvisor := 10000 - Zero_deadband - Full_lever_deadband, Offset := 0);
// Limit ouput to max of 10000
_w7 := LIMIT(0, Linear_abs, 10000);
// Add sign back to the absolute value.
_w9 := SEL(Raw >= 0, Linear_abs, Linear_abs);
// Apply cubic function
_w10 := INT_TO_REAL(Linear);
Cubic := REAL_TO_INT((_w10 * _w10 * _w10) / _w11);
hmi_Data.Status.1 := _w13;
Power_lever_data.Reverse := SEL(Use_neutral, Reverse, _w12 AND NOT Neutral);
_w11 := 10000 * 10000;
Power_lever_data.Neutral := _w14;
// This has been changed to MOVE blocks to set individual bits of the Status word
// as the CFC block for BOOL_TO_WORD does not have 16 inputs for some reason
_w15 := Power_lever_data.Forward;
Power_lever_data.Raw := Raw;
_w17 := SEL(Use_neutral, Forward, _w16);
// Power lever data section
// Pack data in Power_lever_data stucture.
_w16 := Linear > 0 AND NOT Neutral;
Power_lever_data.Forward := _w17;
_w13 := Power_lever_data.Reverse;
_w12 := Linear < 0;
_w14 := _w18 OR _w19;
_w19 := Forward AND Reverse AND Use_neutral;
hmi_Data.Status.0 := _w15;
Power_lever_data.Button := Button;
cs_Forward_and_reverse := _w20;
Power_lever_data.Linear := Linear;
Power_lever_data.Cubic := Cubic;
cs_Pot_fwd_no_notch := TON_0.Q;
_w18 := Neutral AND Use_neutral;
hmi_data.Raw := Raw;
_w21 := Linear;
TON_1(IN := (-Raw) > _w22 AND NOT Reverse, PT := t#500ms); // TON
// Pot shows that lever is reverse but the reverse notch is not activated
_w22 := Notch_position + Allowed_notch_variation;
hmi_data.Linear := _w21;
// Pot is out of range negative
_w23 := Pot < Neg_out_of_range_val;
cs_Pot_rev_no_notch := TON_1.Q;
hmi_data.Cubic := Cubic;
hmi_Data.Status.2 := Power_lever_data.Neutral;
hmi_Data.Status.3 := Button;
// Power lever faults section
// Forward and reverse notches simulateously active
_w20 := Forward AND Reverse;
// Pot shows that lever is forward but the forward notch is not activated
TON_0(IN := Raw > Notch_position + Allowed_notch_variation AND NOT Forward, PT := t#500ms); // TON
cs_Out_of_range_neg := _w23;
TON_2(IN := Raw < _w24 AND Forward, PT := t#500ms); // TON
// Forward notch is activated but the pot does not show that the lever is past the forward notch
_w24 := Notch_position - Allowed_notch_variation;
cs_Fwd_notch_not_pot := TON_2.Q;
TON_3(IN := (-Raw) < _w25 AND Reverse, PT := t#500ms); // TON
// Reverse notch is activated but the pot does not show that the lever is past the reverse notch
_w25 := Notch_position - Allowed_notch_variation;
cs_Rev_notch_not_pot := TON_3.Q;
// Pot is out of range positive
cs_Out_of_range_pos := Pot > Pos_out_of_range_val;
END_METHOD

METHOD Standard_stuff
VAR_INPUT
	Bits_from_hmi:ARRAY[0..1] OF WORD;
	Creep_switch:BOOL;
	Slow_switch:BOOL;
	Normal_switch:BOOL;
	Watchdog_heartbeat:BOOL;
	System_start:BOOL;
	System_stop:BOOL;
	System_started:BOOL;
	SCC:BOOL;
END_VAR
VAR_OUTPUT
	Bits_to_hmi:ARRAY[0..1] OF WORD;
	Hmi_test_trip:BOOL;
	Watchdog_test_0:BOOL;
	Watchdog_test_1:BOOL;
	Activity:BOOL;
END_VAR
VAR_INST // added by the converter: edge detectors and wires of the graphical bodies
    _w1, _w2, _w3, _w4, _w5, _w6 : ANY;
END_VAR
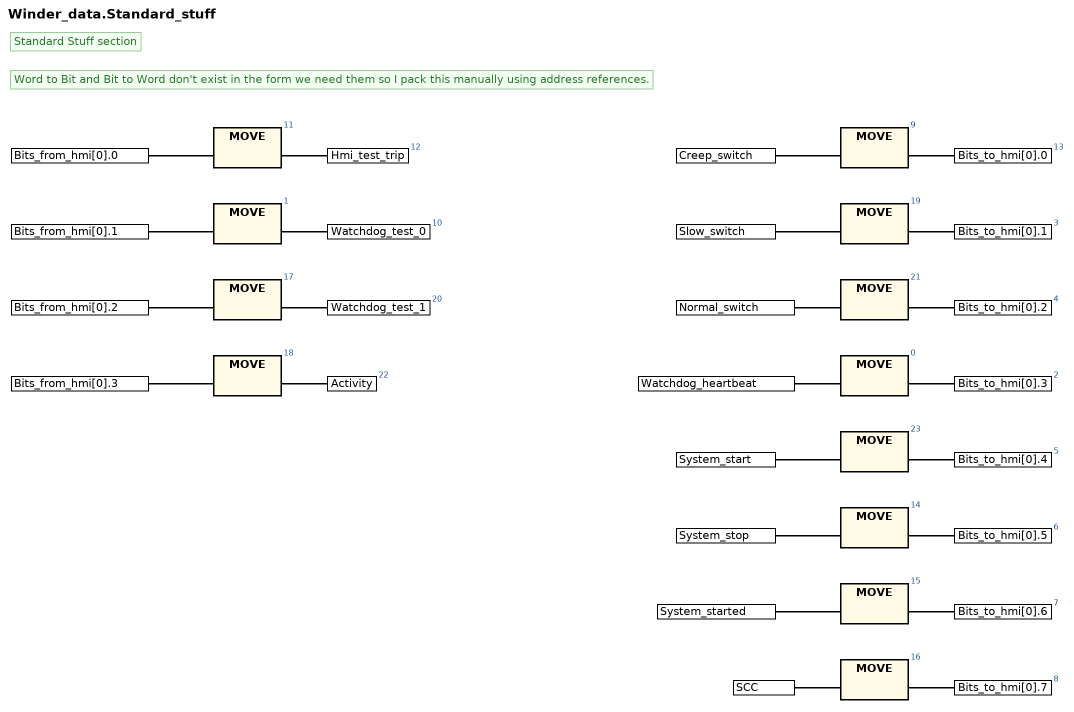
Bits_to_hmi[0].3 := Watchdog_heartbeat;
Bits_to_hmi[0].1 := _w1;
Bits_to_hmi[0].2 := _w2;
Bits_to_hmi[0].4 := _w3;
Bits_to_hmi[0].5 := _w4;
Bits_to_hmi[0].6 := _w5;
Bits_to_hmi[0].7 := _w6;
Watchdog_test_0 := Bits_from_hmi[0].1;
// Standard Stuff section
// Word to Bit and Bit to Word don't exist in the form we need them so I pack this manually using address references.
Hmi_test_trip := Bits_from_hmi[0].0;
Bits_to_hmi[0].0 := Creep_switch;
_w4 := System_stop;
_w5 := System_started;
_w6 := SCC;
_w1 := Slow_switch;
Watchdog_test_1 := Bits_from_hmi[0].2;
_w2 := Normal_switch;
Activity := Bits_from_hmi[0].3;
_w3 := System_start;
END_METHOD

END_PROGRAM

(* stored: Version 1.1.0.1, ProductVersion 3.1.4024.0
   POU Winder_data: Id {adeaff29-a88d-4b52-a1fb-ee7f456997be}, SpecialFunc None
   Method Brake: Id {ed2d8eae-d25a-4268-aa71-9e73c8cfcb7a}
   Method Clutch: Id {510a9873-1d5f-4e7c-bbd1-4609c7ff8320}
   Method Mode: Id {9b1a21d6-1326-46a2-8d44-c677cbf706bd}
   Method Power_lever: Id {e2e72fe3-40f7-4272-8447-d40af7cfaa7e}
   Method Standard_stuff: Id {255362e7-64c4-4c25-9ed0-062a55fc5f2f} *)
